// TIA Portal V20 export
VAR_GLOBAL   // PLC tag table "LER_LIU117"
END_VAR
VAR_GLOBAL CONSTANT   // user constants
   LIU117_Lengths : Int := 2;
END_VAR
